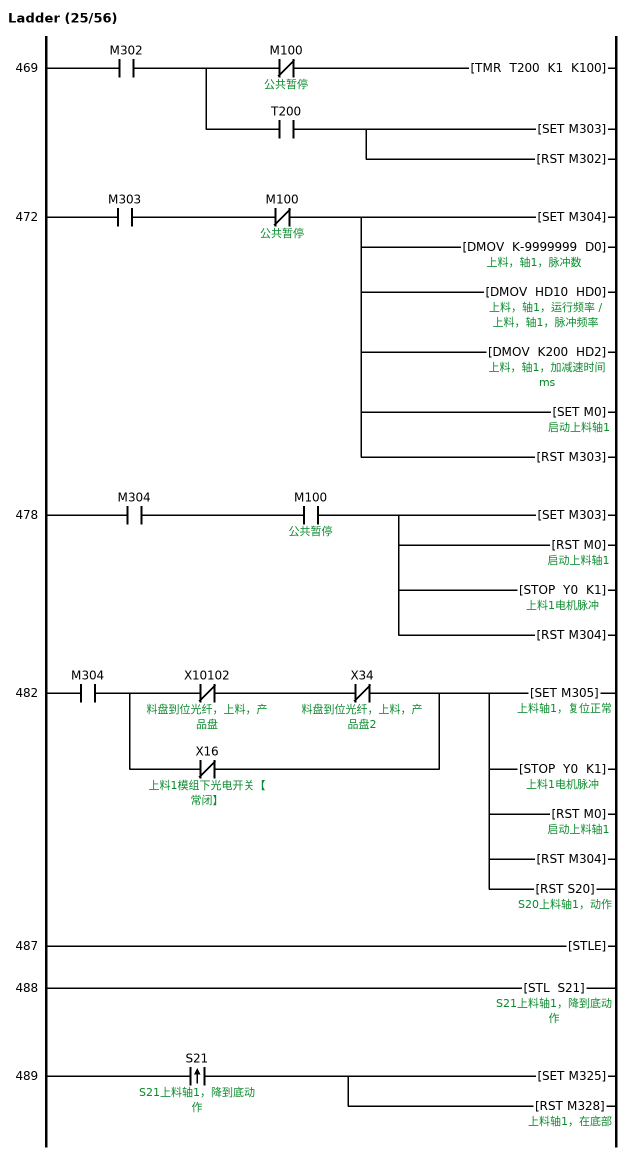
[picture p24: Ladder rows 469-489]
LD     M302
MPS
ANI    M100	; 公共暂停
TMR    T200 K1 K100
MPP
AND    T200
SET    M303
RST    M302
LD     M303
ANI    M100	; 公共暂停
SET    M304
DMOV   K-9999999 D0	; 上料，轴1，脉冲数
DMOV   HD10 HD0	; 上料，轴1，运行频率 / 上料，轴1，脉冲频率
DMOV   K200 HD2	; 上料，轴1，加减速时间ms
SET    M0	; 启动上料轴1
RST    M303
LD     M304
AND    M100	; 公共暂停
SET    M303
RST    M0	; 启动上料轴1
STOP   Y0 K1	; 上料1电机脉冲
RST    M304
LD     M304
LDI    X10102	; 料盘到位光纤，上料，产品盘
ANI    X34	; 料盘到位光纤，上料，产品盘2
ORI    X16	; 上料1模组下光电开关【常闭】
ANB
SET    M305	; 上料轴1，复位正常
STOP   Y0 K1	; 上料1电机脉冲
RST    M0	; 启动上料轴1
RST    M304
RST    S20	; S20上料轴1，动作
STLE
STL    S21	; S21上料轴1，降到底动作
LDP    S21	; S21上料轴1，降到底动作
SET    M325
RST    M328	; 上料轴1，在底部

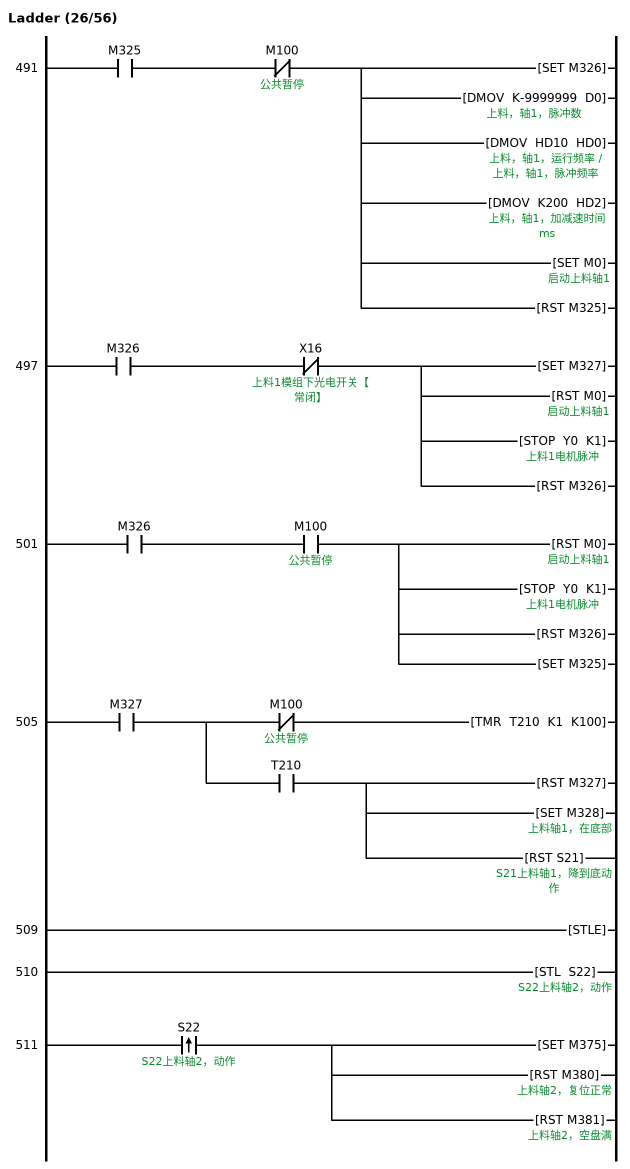
LD     M325
ANI    M100	; 公共暂停
SET    M326
DMOV   K-9999999 D0	; 上料，轴1，脉冲数
DMOV   HD10 HD0	; 上料，轴1，运行频率 / 上料，轴1，脉冲频率
DMOV   K200 HD2	; 上料，轴1，加减速时间ms
SET    M0	; 启动上料轴1
RST    M325
LD     M326
ANI    X16	; 上料1模组下光电开关【常闭】
SET    M327
RST    M0	; 启动上料轴1
STOP   Y0 K1	; 上料1电机脉冲
RST    M326
LD     M326
AND    M100	; 公共暂停
RST    M0	; 启动上料轴1
STOP   Y0 K1	; 上料1电机脉冲
RST    M326
SET    M325
LD     M327
MPS
ANI    M100	; 公共暂停
TMR    T210 K1 K100
MPP
AND    T210
RST    M327
SET    M328	; 上料轴1，在底部
RST    S21	; S21上料轴1，降到底动作
STLE
STL    S22	; S22上料轴2，动作
LDP    S22	; S22上料轴2，动作
SET    M375
RST    M380	; 上料轴2，复位正常
RST    M381	; 上料轴2，空盘满

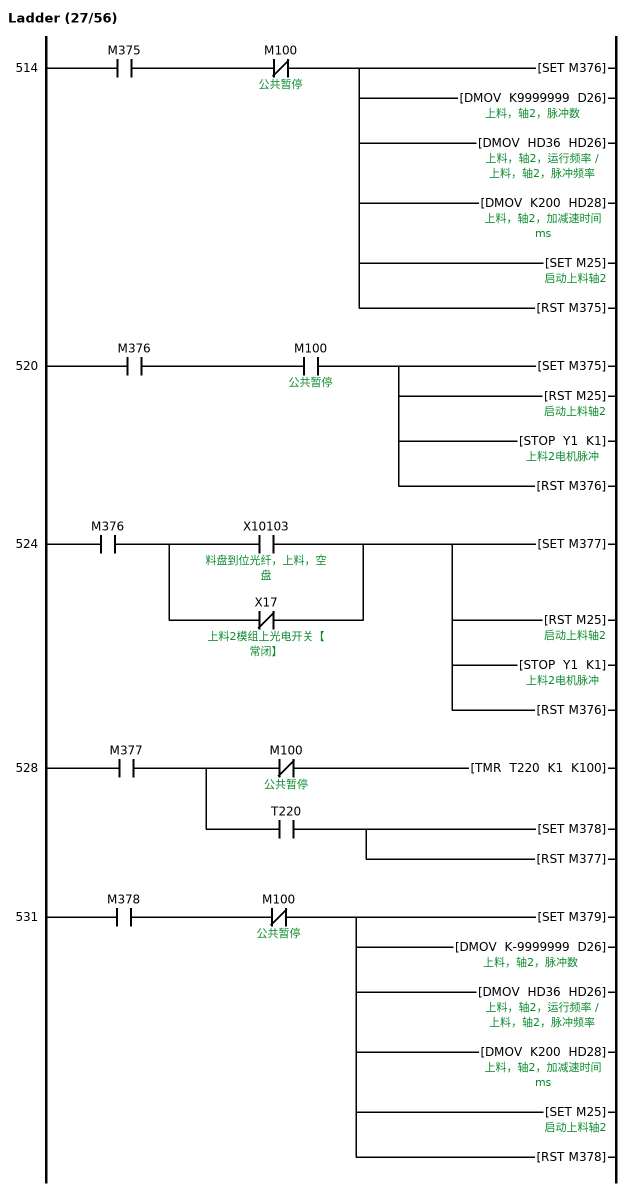
LD     M375
ANI    M100	; 公共暂停
SET    M376
DMOV   K9999999 D26	; 上料，轴2，脉冲数
DMOV   HD36 HD26	; 上料，轴2，运行频率 / 上料，轴2，脉冲频率
DMOV   K200 HD28	; 上料，轴2，加减速时间ms
SET    M25	; 启动上料轴2
RST    M375
LD     M376
AND    M100	; 公共暂停
SET    M375
RST    M25	; 启动上料轴2
STOP   Y1 K1	; 上料2电机脉冲
RST    M376
LD     M376
LD     X10103	; 料盘到位光纤，上料，空盘
ORI    X17	; 上料2模组上光电开关【常闭】
ANB
SET    M377
RST    M25	; 启动上料轴2
STOP   Y1 K1	; 上料2电机脉冲
RST    M376
LD     M377
MPS
ANI    M100	; 公共暂停
TMR    T220 K1 K100
MPP
AND    T220
SET    M378
RST    M377
LD     M378
ANI    M100	; 公共暂停
SET    M379
DMOV   K-9999999 D26	; 上料，轴2，脉冲数
DMOV   HD36 HD26	; 上料，轴2，运行频率 / 上料，轴2，脉冲频率
DMOV   K200 HD28	; 上料，轴2，加减速时间ms
SET    M25	; 启动上料轴2
RST    M378

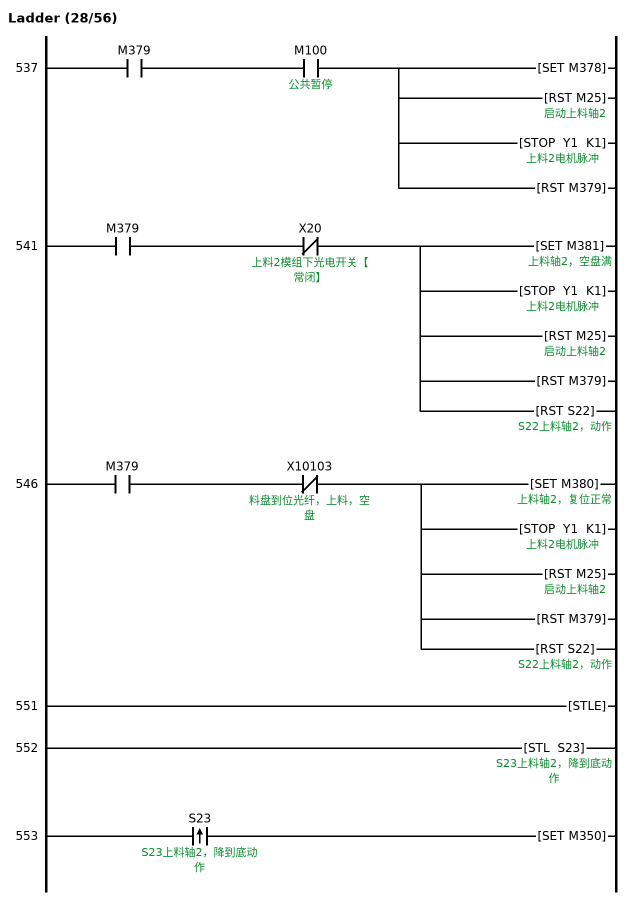
LD     M379
AND    M100	; 公共暂停
SET    M378
RST    M25	; 启动上料轴2
STOP   Y1 K1	; 上料2电机脉冲
RST    M379
LD     M379
ANI    X20	; 上料2模组下光电开关【常闭】
SET    M381	; 上料轴2，空盘满
STOP   Y1 K1	; 上料2电机脉冲
RST    M25	; 启动上料轴2
RST    M379
RST    S22	; S22上料轴2，动作
LD     M379
ANI    X10103	; 料盘到位光纤，上料，空盘
SET    M380	; 上料轴2，复位正常
STOP   Y1 K1	; 上料2电机脉冲
RST    M25	; 启动上料轴2
RST    M379
RST    S22	; S22上料轴2，动作
STLE
STL    S23	; S23上料轴2，降到底动作
LDP    S23	; S23上料轴2，降到底动作
SET    M350

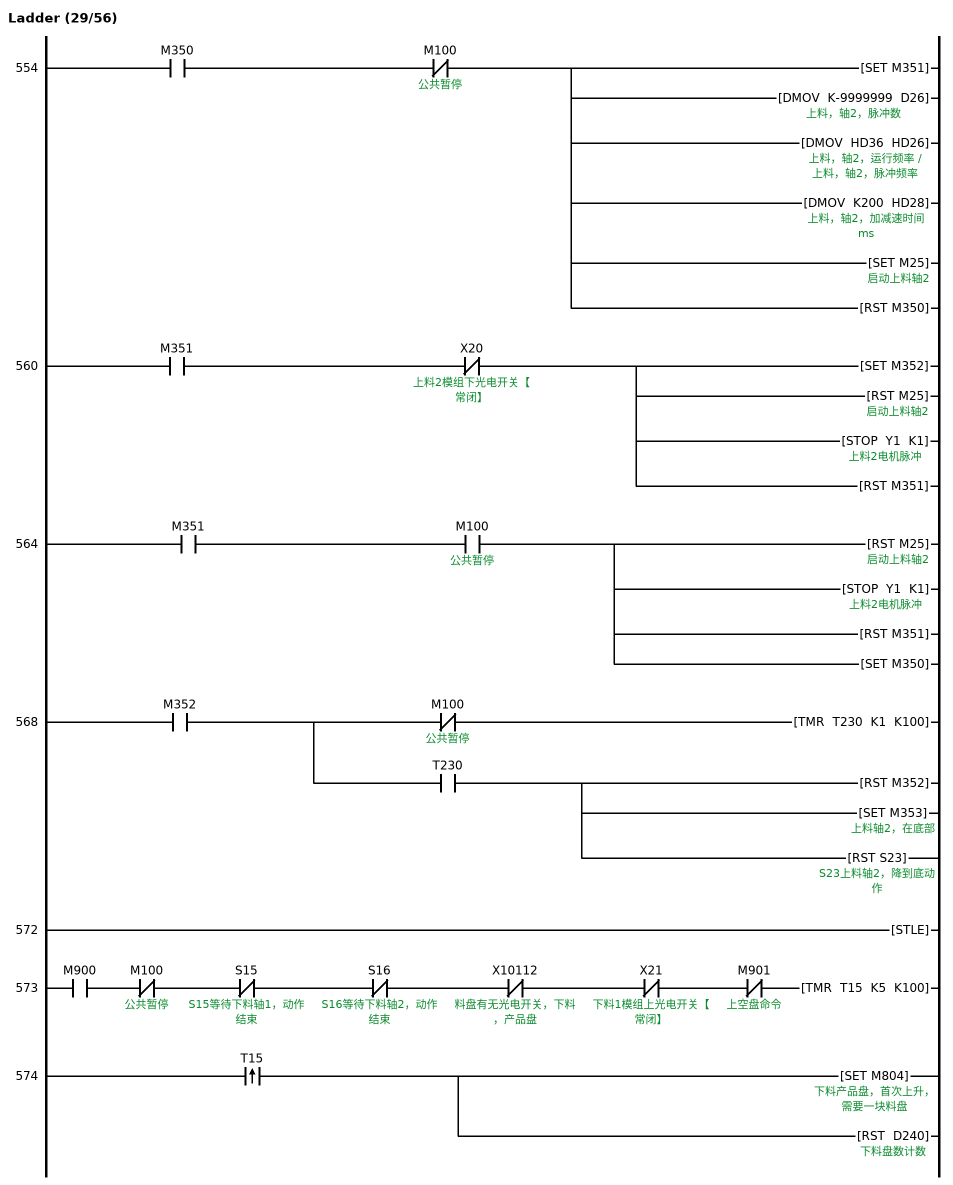
LD     M350
ANI    M100	; 公共暂停
SET    M351
DMOV   K-9999999 D26	; 上料，轴2，脉冲数
DMOV   HD36 HD26	; 上料，轴2，运行频率 / 上料，轴2，脉冲频率
DMOV   K200 HD28	; 上料，轴2，加减速时间ms
SET    M25	; 启动上料轴2
RST    M350
LD     M351
ANI    X20	; 上料2模组下光电开关【常闭】
SET    M352
RST    M25	; 启动上料轴2
STOP   Y1 K1	; 上料2电机脉冲
RST    M351
LD     M351
AND    M100	; 公共暂停
RST    M25	; 启动上料轴2
STOP   Y1 K1	; 上料2电机脉冲
RST    M351
SET    M350
LD     M352
MPS
ANI    M100	; 公共暂停
TMR    T230 K1 K100
MPP
AND    T230
RST    M352
SET    M353	; 上料轴2，在底部
RST    S23	; S23上料轴2，降到底动作
STLE
LD     M900
ANI    M100	; 公共暂停
ANI    S15	; S15等待下料轴1，动作结束
ANI    S16	; S16等待下料轴2，动作结束
ANI    X10112	; 料盘有无光电开关，下料，产品盘
ANI    X21	; 下料1模组上光电开关【常闭】
ANI    M901	; 上空盘命令
TMR    T15 K5 K100
LDP    T15
SET    M804	; 下料产品盘，首次上升，需要一块料盘
RST    D240	; 下料盘数计数

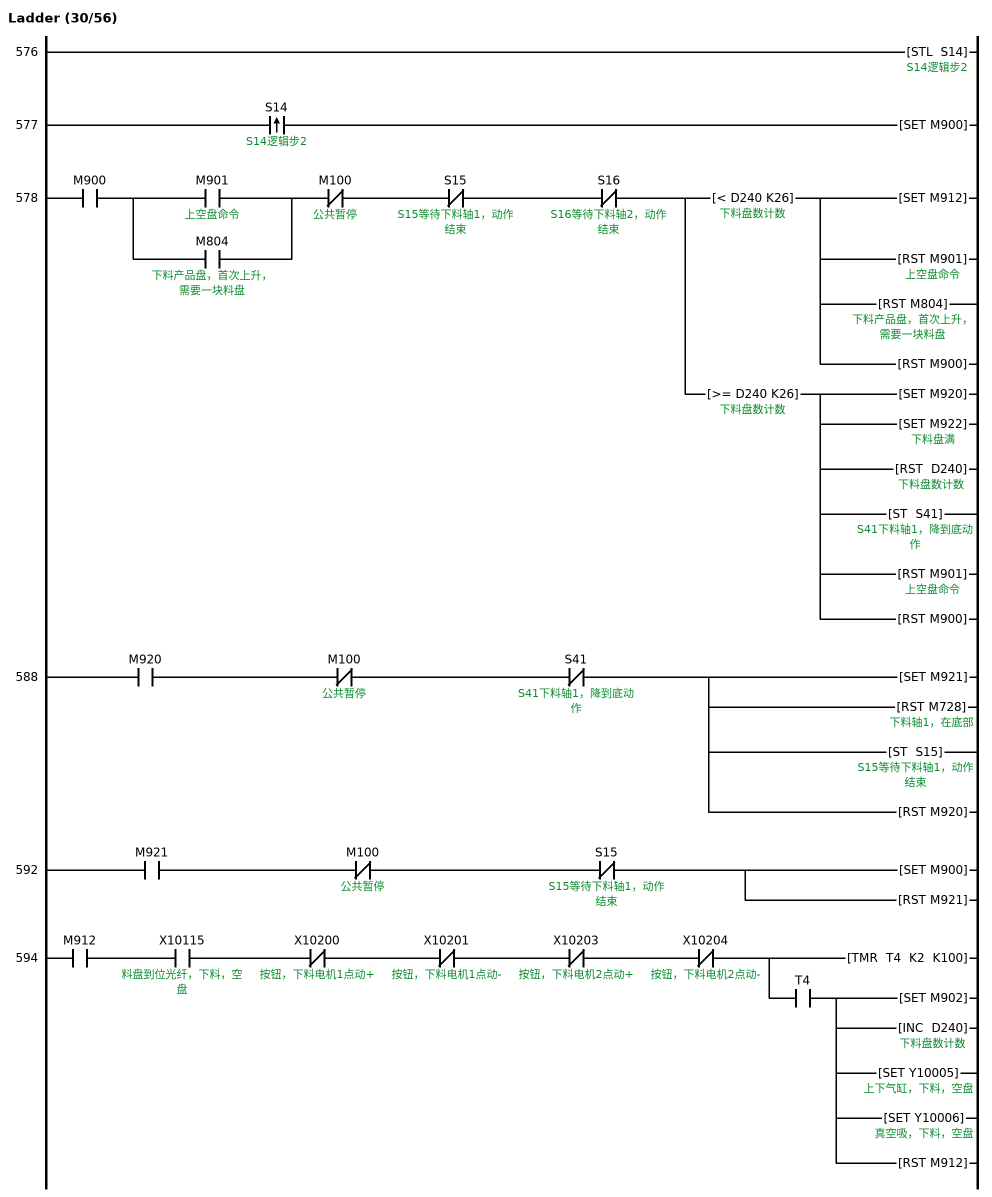
STL    S14	; S14逻辑步2
LDP    S14	; S14逻辑步2
SET    M900
LD     M900
LD     M901	; 上空盘命令
OR     M804	; 下料产品盘，首次上升，需要一块料盘
ANB
ANI    M100	; 公共暂停
ANI    S15	; S15等待下料轴1，动作结束
ANI    S16	; S16等待下料轴2，动作结束
MPS
AND<   D240 K26	; 下料盘数计数
SET    M912
RST    M901	; 上空盘命令
RST    M804	; 下料产品盘，首次上升，需要一块料盘
RST    M900
MPP
AND>=  D240 K26	; 下料盘数计数
SET    M920
SET    M922	; 下料盘满
RST    D240	; 下料盘数计数
ST     S41	; S41下料轴1，降到底动作
RST    M901	; 上空盘命令
RST    M900
LD     M920
ANI    M100	; 公共暂停
ANI    S41	; S41下料轴1，降到底动作
SET    M921
RST    M728	; 下料轴1，在底部
ST     S15	; S15等待下料轴1，动作结束
RST    M920
LD     M921
ANI    M100	; 公共暂停
ANI    S15	; S15等待下料轴1，动作结束
SET    M900
RST    M921
LD     M912
AND    X10115	; 料盘到位光纤，下料，空盘
ANI    X10200	; 按钮，下料电机1点动+
ANI    X10201	; 按钮，下料电机1点动-
ANI    X10203	; 按钮，下料电机2点动+
ANI    X10204	; 按钮，下料电机2点动-
TMR    T4 K2 K100
AND    T4
SET    M902
INC    D240	; 下料盘数计数
SET    Y10005	; 上下气缸，下料，空盘
SET    Y10006	; 真空吸，下料，空盘
RST    M912

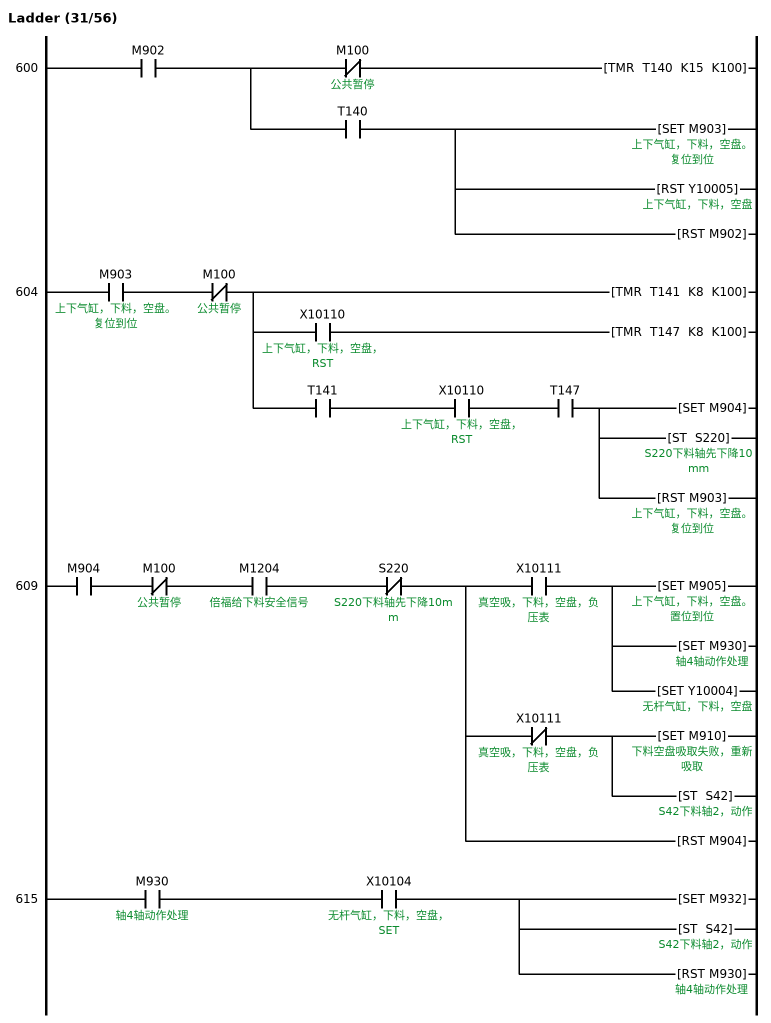
LD     M902
MPS
ANI    M100	; 公共暂停
TMR    T140 K15 K100
MPP
AND    T140
SET    M903	; 上下气缸，下料，空盘。复位到位
RST    Y10005	; 上下气缸，下料，空盘
RST    M902
LD     M903	; 上下气缸，下料，空盘。复位到位
ANI    M100	; 公共暂停
TMR    T141 K8 K100
MPS
AND    X10110	; 上下气缸，下料，空盘，RST
TMR    T147 K8 K100
MPP
AND    T141
AND    X10110	; 上下气缸，下料，空盘，RST
AND    T147
SET    M904
ST     S220	; S220下料轴先下降10mm
RST    M903	; 上下气缸，下料，空盘。复位到位
LD     M904
ANI    M100	; 公共暂停
AND    M1204	; 倍福给下料安全信号
ANI    S220	; S220下料轴先下降10mm
MPS
AND    X10111	; 真空吸，下料，空盘，负压表
SET    M905	; 上下气缸，下料，空盘。置位到位
SET    M930	; 轴4轴动作处理
SET    Y10004	; 无杆气缸，下料，空盘
MRD
ANI    X10111	; 真空吸，下料，空盘，负压表
SET    M910	; 下料空盘吸取失败，重新吸取
ST     S42	; S42下料轴2，动作
MPP
RST    M904
LD     M930	; 轴4轴动作处理
AND    X10104	; 无杆气缸，下料，空盘，SET
SET    M932
ST     S42	; S42下料轴2，动作
RST    M930	; 轴4轴动作处理

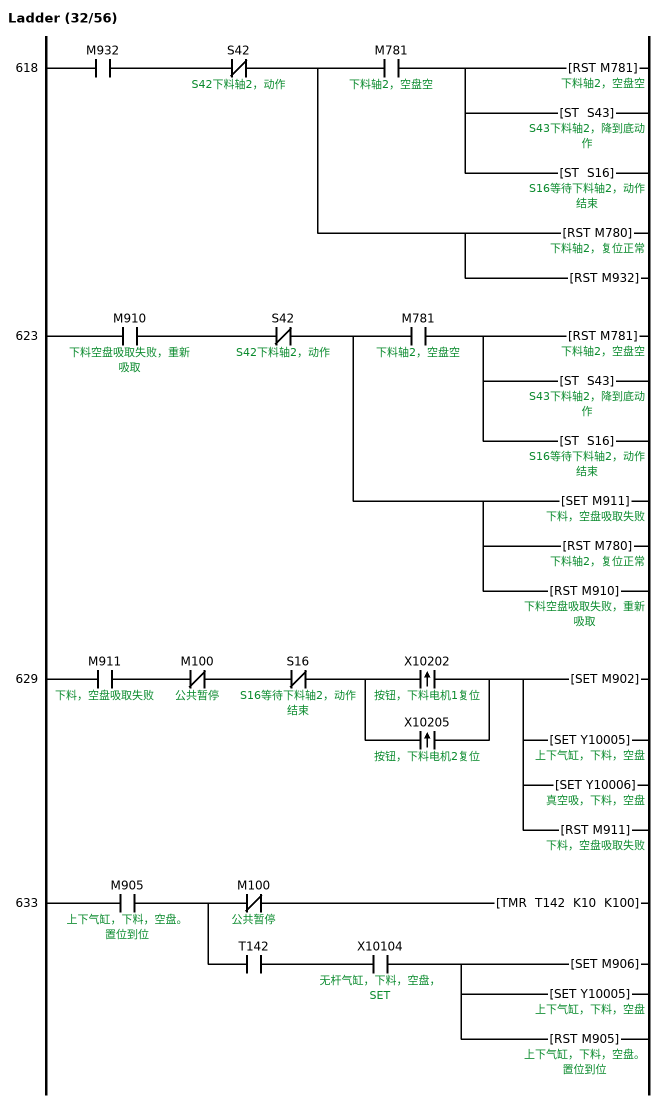
LD     M932
ANI    S42	; S42下料轴2，动作
MPS
AND    M781	; 下料轴2，空盘空
RST    M781	; 下料轴2，空盘空
ST     S43	; S43下料轴2，降到底动作
ST     S16	; S16等待下料轴2，动作结束
MPP
RST    M780	; 下料轴2，复位正常
RST    M932
LD     M910	; 下料空盘吸取失败，重新吸取
ANI    S42	; S42下料轴2，动作
MPS
AND    M781	; 下料轴2，空盘空
RST    M781	; 下料轴2，空盘空
ST     S43	; S43下料轴2，降到底动作
ST     S16	; S16等待下料轴2，动作结束
MPP
SET    M911	; 下料，空盘吸取失败
RST    M780	; 下料轴2，复位正常
RST    M910	; 下料空盘吸取失败，重新吸取
LD     M911	; 下料，空盘吸取失败
ANI    M100	; 公共暂停
ANI    S16	; S16等待下料轴2，动作结束
LDP    X10202	; 按钮，下料电机1复位
ORP    X10205	; 按钮，下料电机2复位
ANB
SET    M902
SET    Y10005	; 上下气缸，下料，空盘
SET    Y10006	; 真空吸，下料，空盘
RST    M911	; 下料，空盘吸取失败
LD     M905	; 上下气缸，下料，空盘。置位到位
MPS
ANI    M100	; 公共暂停
TMR    T142 K10 K100
MPP
AND    T142
AND    X10104	; 无杆气缸，下料，空盘，SET
SET    M906
SET    Y10005	; 上下气缸，下料，空盘
RST    M905	; 上下气缸，下料，空盘。置位到位

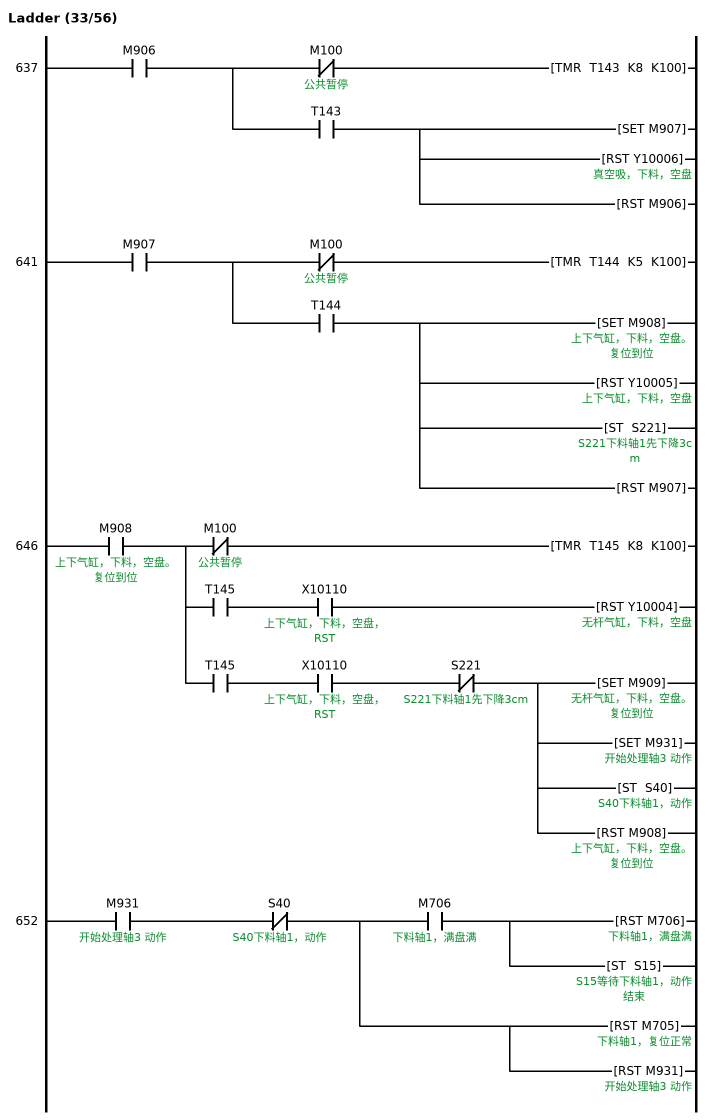
LD     M906
MPS
ANI    M100	; 公共暂停
TMR    T143 K8 K100
MPP
AND    T143
SET    M907
RST    Y10006	; 真空吸，下料，空盘
RST    M906
LD     M907
MPS
ANI    M100	; 公共暂停
TMR    T144 K5 K100
MPP
AND    T144
SET    M908	; 上下气缸，下料，空盘。复位到位
RST    Y10005	; 上下气缸，下料，空盘
ST     S221	; S221下料轴1先下降3cm
RST    M907
LD     M908	; 上下气缸，下料，空盘。复位到位
MPS
ANI    M100	; 公共暂停
TMR    T145 K8 K100
MRD
AND    T145
AND    X10110	; 上下气缸，下料，空盘，RST
RST    Y10004	; 无杆气缸，下料，空盘
MPP
AND    T145
AND    X10110	; 上下气缸，下料，空盘，RST
ANI    S221	; S221下料轴1先下降3cm
SET    M909	; 无杆气缸，下料，空盘。复位到位
SET    M931	; 开始处理轴3 动作
ST     S40	; S40下料轴1，动作
RST    M908	; 上下气缸，下料，空盘。复位到位
LD     M931	; 开始处理轴3 动作
ANI    S40	; S40下料轴1，动作
MPS
AND    M706	; 下料轴1，满盘满
RST    M706	; 下料轴1，满盘满
ST     S15	; S15等待下料轴1，动作结束
MPP
RST    M705	; 下料轴1，复位正常
RST    M931	; 开始处理轴3 动作

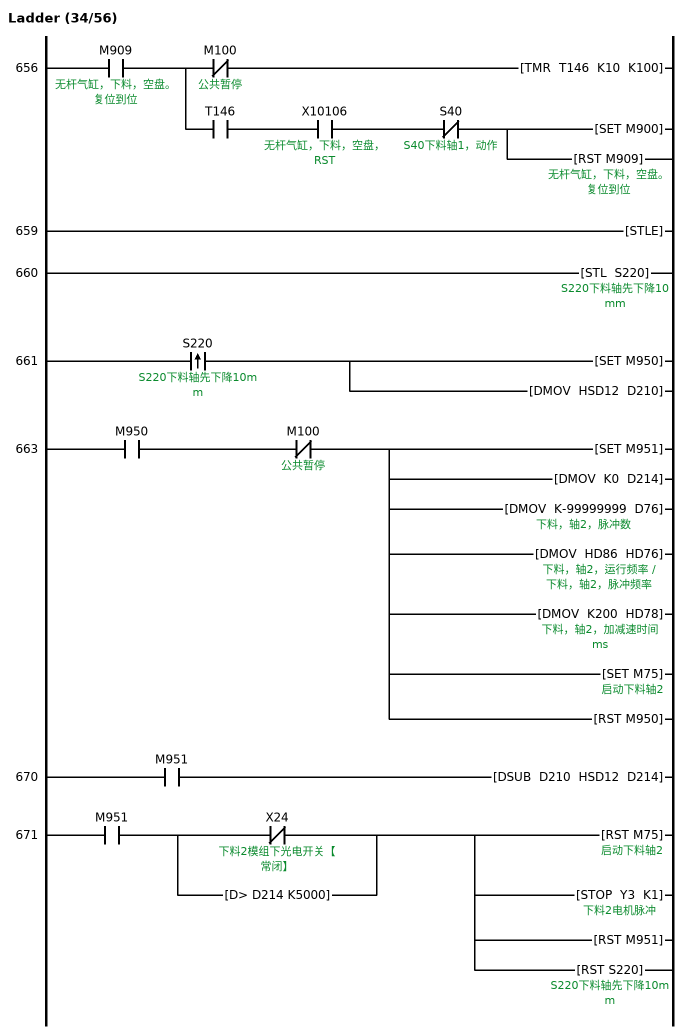
LD     M909	; 无杆气缸，下料，空盘。复位到位
MPS
ANI    M100	; 公共暂停
TMR    T146 K10 K100
MPP
AND    T146
AND    X10106	; 无杆气缸，下料，空盘，RST
ANI    S40	; S40下料轴1，动作
SET    M900
RST    M909	; 无杆气缸，下料，空盘。复位到位
STLE
STL    S220	; S220下料轴先下降10mm
LDP    S220	; S220下料轴先下降10mm
SET    M950
DMOV   HSD12 D210
LD     M950
ANI    M100	; 公共暂停
SET    M951
DMOV   K0 D214
DMOV   K-99999999 D76	; 下料，轴2，脉冲数
DMOV   HD86 HD76	; 下料，轴2，运行频率 / 下料，轴2，脉冲频率
DMOV   K200 HD78	; 下料，轴2，加减速时间ms
SET    M75	; 启动下料轴2
RST    M950
LD     M951
DSUB   D210 HSD12 D214
LD     M951
LDI    X24	; 下料2模组下光电开关【常闭】
DOR>   D214 K5000
ANB
RST    M75	; 启动下料轴2
STOP   Y3 K1	; 下料2电机脉冲
RST    M951
RST    S220	; S220下料轴先下降10mm

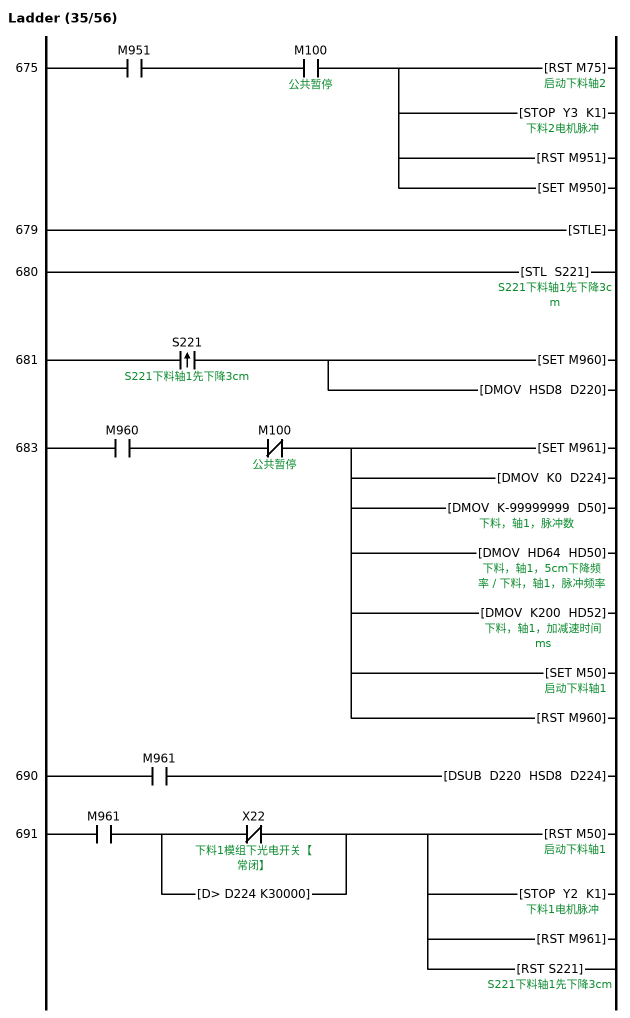
LD     M951
AND    M100	; 公共暂停
RST    M75	; 启动下料轴2
STOP   Y3 K1	; 下料2电机脉冲
RST    M951
SET    M950
STLE
STL    S221	; S221下料轴1先下降3cm
LDP    S221	; S221下料轴1先下降3cm
SET    M960
DMOV   HSD8 D220
LD     M960
ANI    M100	; 公共暂停
SET    M961
DMOV   K0 D224
DMOV   K-99999999 D50	; 下料，轴1，脉冲数
DMOV   HD64 HD50	; 下料，轴1，5cm下降频率 / 下料，轴1，脉冲频率
DMOV   K200 HD52	; 下料，轴1，加减速时间ms
SET    M50	; 启动下料轴1
RST    M960
LD     M961
DSUB   D220 HSD8 D224
LD     M961
LDI    X22	; 下料1模组下光电开关【常闭】
DOR>   D224 K30000
ANB
RST    M50	; 启动下料轴1
STOP   Y2 K1	; 下料1电机脉冲
RST    M961
RST    S221	; S221下料轴1先下降3cm

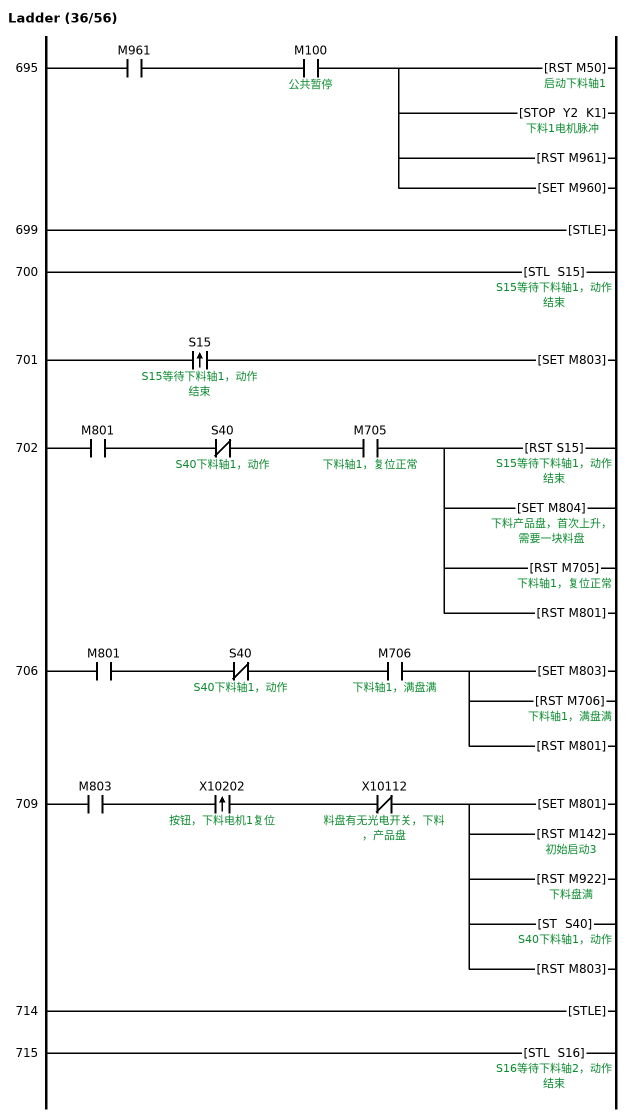
LD     M961
AND    M100	; 公共暂停
RST    M50	; 启动下料轴1
STOP   Y2 K1	; 下料1电机脉冲
RST    M961
SET    M960
STLE
STL    S15	; S15等待下料轴1，动作结束
LDP    S15	; S15等待下料轴1，动作结束
SET    M803
LD     M801
ANI    S40	; S40下料轴1，动作
AND    M705	; 下料轴1，复位正常
RST    S15	; S15等待下料轴1，动作结束
SET    M804	; 下料产品盘，首次上升，需要一块料盘
RST    M705	; 下料轴1，复位正常
RST    M801
LD     M801
ANI    S40	; S40下料轴1，动作
AND    M706	; 下料轴1，满盘满
SET    M803
RST    M706	; 下料轴1，满盘满
RST    M801
LD     M803
ANDP   X10202	; 按钮，下料电机1复位
ANI    X10112	; 料盘有无光电开关，下料，产品盘
SET    M801
RST    M142	; 初始启动3
RST    M922	; 下料盘满
ST     S40	; S40下料轴1，动作
RST    M803
STLE
STL    S16	; S16等待下料轴2，动作结束

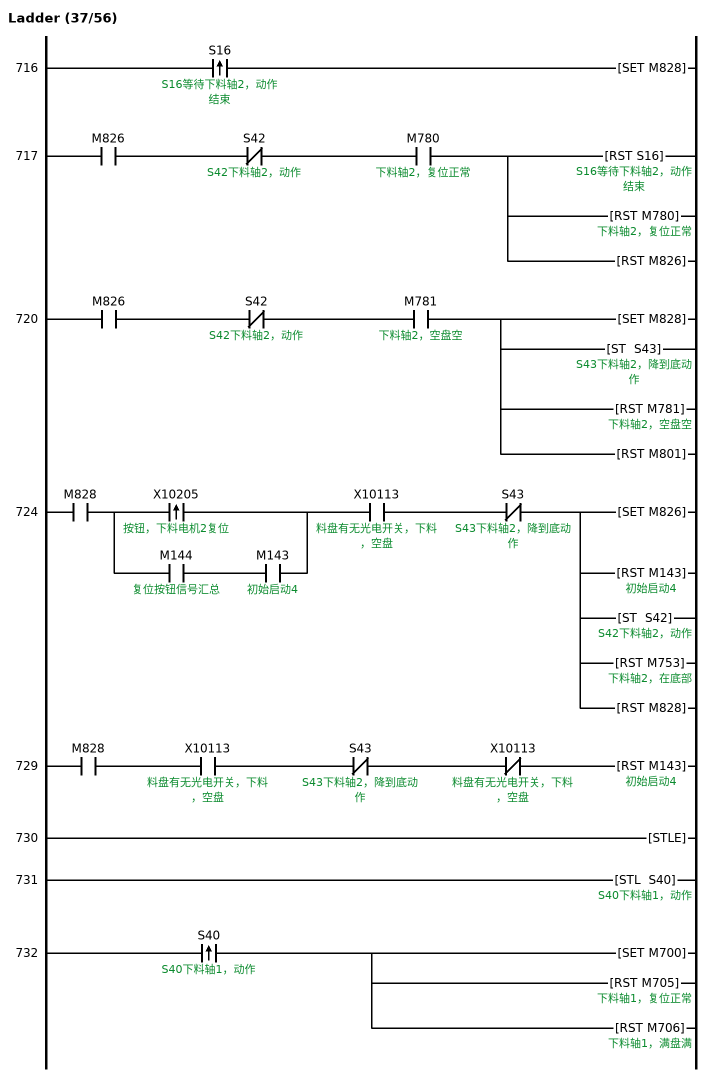
LDP    S16	; S16等待下料轴2，动作结束
SET    M828
LD     M826
ANI    S42	; S42下料轴2，动作
AND    M780	; 下料轴2，复位正常
RST    S16	; S16等待下料轴2，动作结束
RST    M780	; 下料轴2，复位正常
RST    M826
LD     M826
ANI    S42	; S42下料轴2，动作
AND    M781	; 下料轴2，空盘空
SET    M828
ST     S43	; S43下料轴2，降到底动作
RST    M781	; 下料轴2，空盘空
RST    M801
LD     M828
LDP    X10205	; 按钮，下料电机2复位
LD     M144	; 复位按钮信号汇总
AND    M143	; 初始启动4
ORB
ANB
AND    X10113	; 料盘有无光电开关，下料，空盘
ANI    S43	; S43下料轴2，降到底动作
SET    M826
RST    M143	; 初始启动4
ST     S42	; S42下料轴2，动作
RST    M753	; 下料轴2，在底部
RST    M828
LD     M828
AND    X10113	; 料盘有无光电开关，下料，空盘
ANI    S43	; S43下料轴2，降到底动作
ANI    X10113	; 料盘有无光电开关，下料，空盘
RST    M143	; 初始启动4
STLE
STL    S40	; S40下料轴1，动作
LDP    S40	; S40下料轴1，动作
SET    M700
RST    M705	; 下料轴1，复位正常
RST    M706	; 下料轴1，满盘满

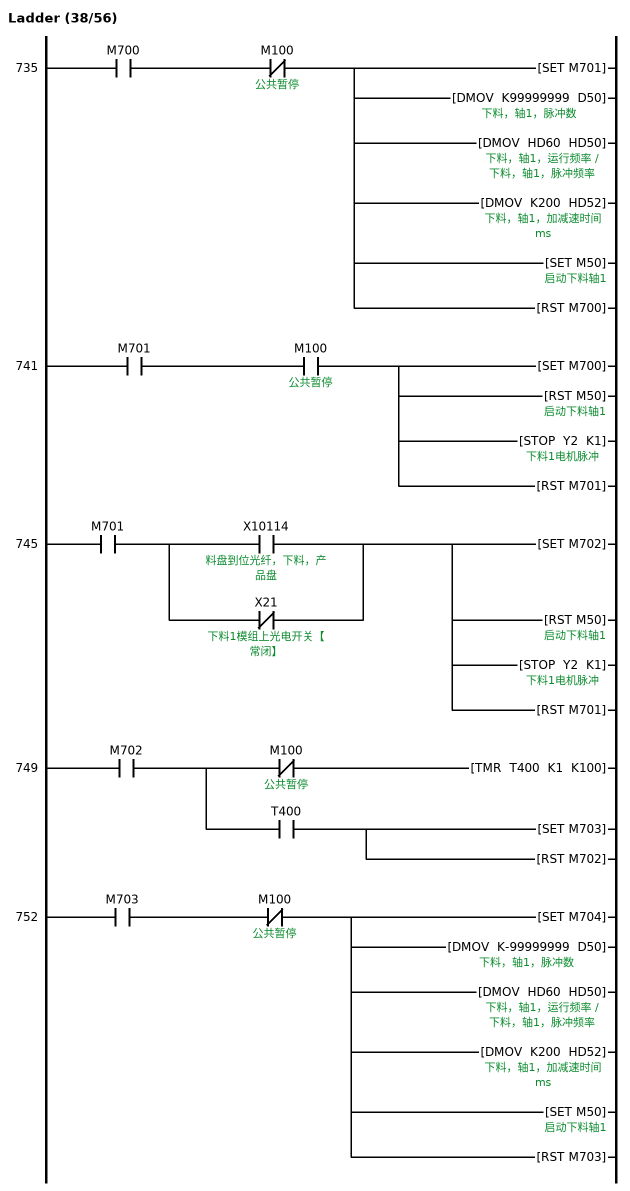
LD     M700
ANI    M100	; 公共暂停
SET    M701
DMOV   K99999999 D50	; 下料，轴1，脉冲数
DMOV   HD60 HD50	; 下料，轴1，运行频率 / 下料，轴1，脉冲频率
DMOV   K200 HD52	; 下料，轴1，加减速时间ms
SET    M50	; 启动下料轴1
RST    M700
LD     M701
AND    M100	; 公共暂停
SET    M700
RST    M50	; 启动下料轴1
STOP   Y2 K1	; 下料1电机脉冲
RST    M701
LD     M701
LD     X10114	; 料盘到位光纤，下料，产品盘
ORI    X21	; 下料1模组上光电开关【常闭】
ANB
SET    M702
RST    M50	; 启动下料轴1
STOP   Y2 K1	; 下料1电机脉冲
RST    M701
LD     M702
MPS
ANI    M100	; 公共暂停
TMR    T400 K1 K100
MPP
AND    T400
SET    M703
RST    M702
LD     M703
ANI    M100	; 公共暂停
SET    M704
DMOV   K-99999999 D50	; 下料，轴1，脉冲数
DMOV   HD60 HD50	; 下料，轴1，运行频率 / 下料，轴1，脉冲频率
DMOV   K200 HD52	; 下料，轴1，加减速时间ms
SET    M50	; 启动下料轴1
RST    M703

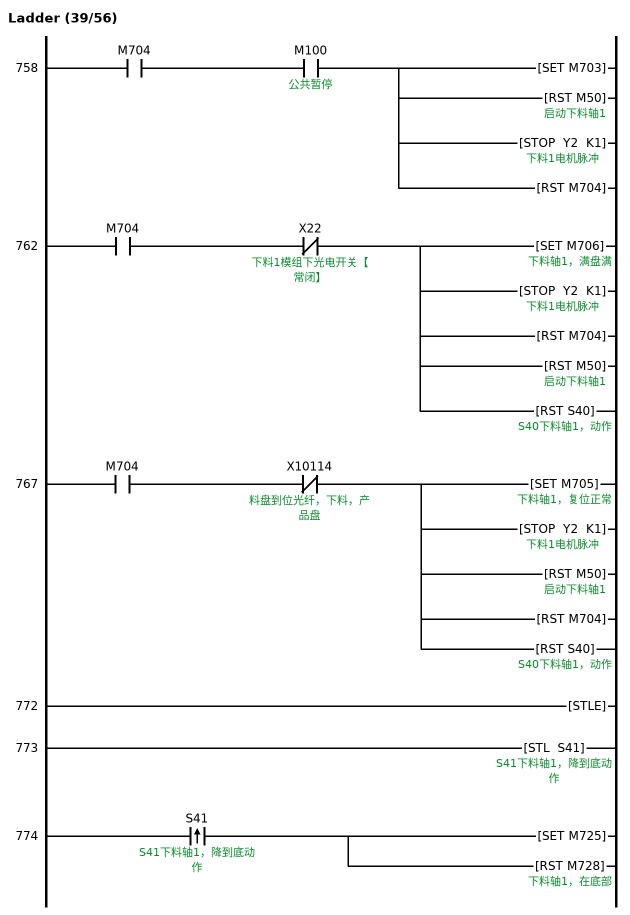
LD     M704
AND    M100	; 公共暂停
SET    M703
RST    M50	; 启动下料轴1
STOP   Y2 K1	; 下料1电机脉冲
RST    M704
LD     M704
ANI    X22	; 下料1模组下光电开关【常闭】
SET    M706	; 下料轴1，满盘满
STOP   Y2 K1	; 下料1电机脉冲
RST    M704
RST    M50	; 启动下料轴1
RST    S40	; S40下料轴1，动作
LD     M704
ANI    X10114	; 料盘到位光纤，下料，产品盘
SET    M705	; 下料轴1，复位正常
STOP   Y2 K1	; 下料1电机脉冲
RST    M50	; 启动下料轴1
RST    M704
RST    S40	; S40下料轴1，动作
STLE
STL    S41	; S41下料轴1，降到底动作
LDP    S41	; S41下料轴1，降到底动作
SET    M725
RST    M728	; 下料轴1，在底部

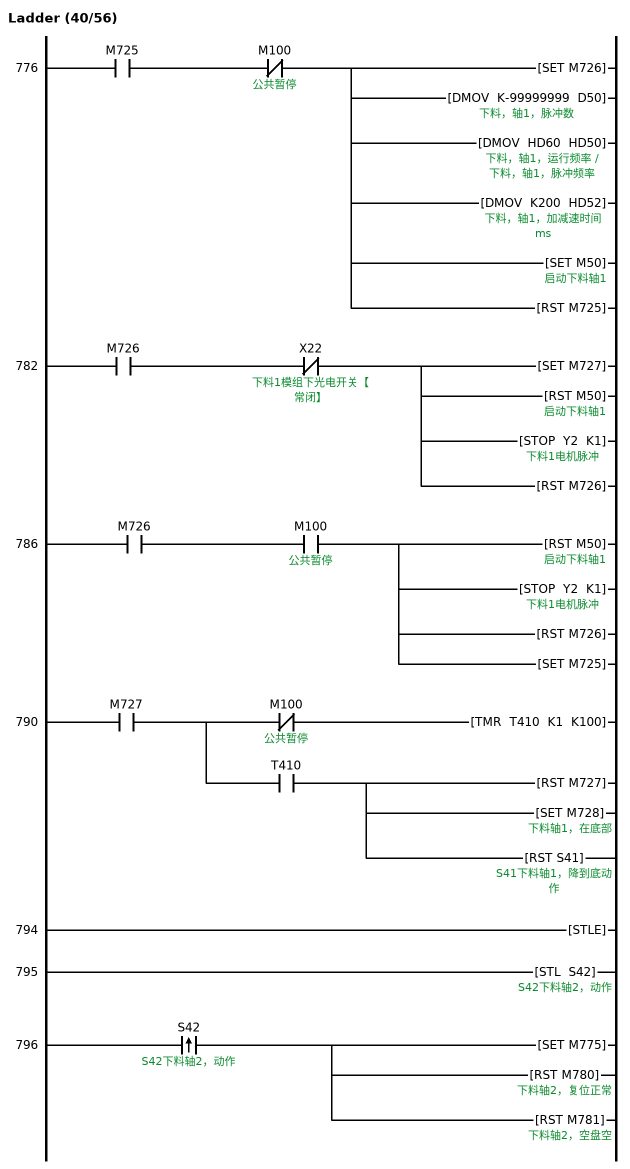
LD     M725
ANI    M100	; 公共暂停
SET    M726
DMOV   K-99999999 D50	; 下料，轴1，脉冲数
DMOV   HD60 HD50	; 下料，轴1，运行频率 / 下料，轴1，脉冲频率
DMOV   K200 HD52	; 下料，轴1，加减速时间ms
SET    M50	; 启动下料轴1
RST    M725
LD     M726
ANI    X22	; 下料1模组下光电开关【常闭】
SET    M727
RST    M50	; 启动下料轴1
STOP   Y2 K1	; 下料1电机脉冲
RST    M726
LD     M726
AND    M100	; 公共暂停
RST    M50	; 启动下料轴1
STOP   Y2 K1	; 下料1电机脉冲
RST    M726
SET    M725
LD     M727
MPS
ANI    M100	; 公共暂停
TMR    T410 K1 K100
MPP
AND    T410
RST    M727
SET    M728	; 下料轴1，在底部
RST    S41	; S41下料轴1，降到底动作
STLE
STL    S42	; S42下料轴2，动作
LDP    S42	; S42下料轴2，动作
SET    M775
RST    M780	; 下料轴2，复位正常
RST    M781	; 下料轴2，空盘空

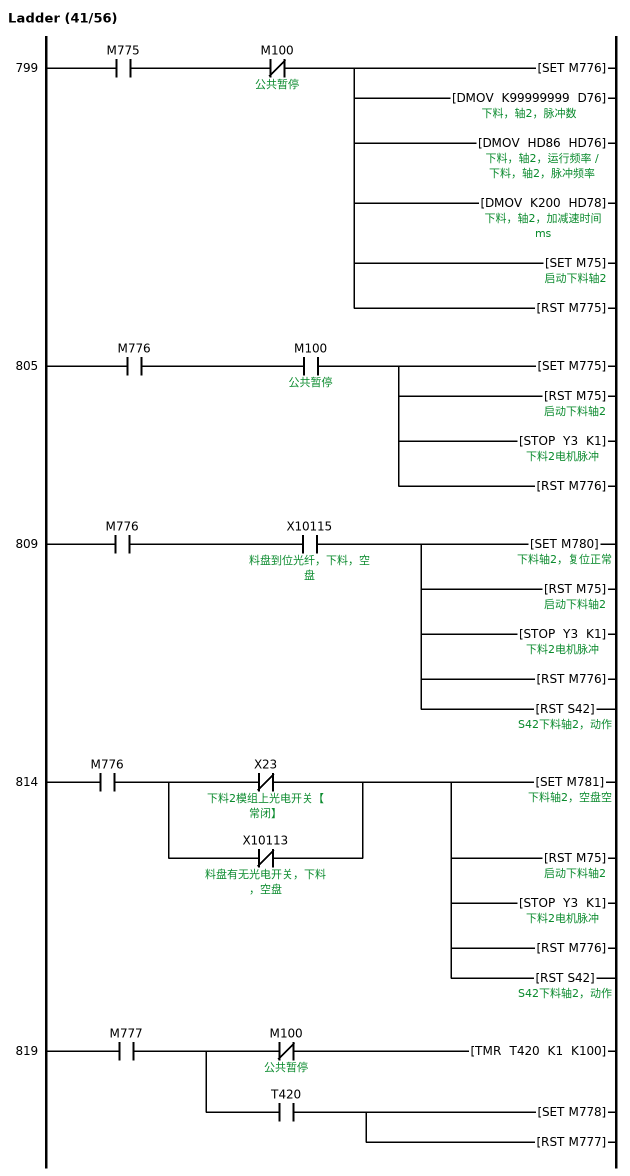
LD     M775
ANI    M100	; 公共暂停
SET    M776
DMOV   K99999999 D76	; 下料，轴2，脉冲数
DMOV   HD86 HD76	; 下料，轴2，运行频率 / 下料，轴2，脉冲频率
DMOV   K200 HD78	; 下料，轴2，加减速时间ms
SET    M75	; 启动下料轴2
RST    M775
LD     M776
AND    M100	; 公共暂停
SET    M775
RST    M75	; 启动下料轴2
STOP   Y3 K1	; 下料2电机脉冲
RST    M776
LD     M776
AND    X10115	; 料盘到位光纤，下料，空盘
SET    M780	; 下料轴2，复位正常
RST    M75	; 启动下料轴2
STOP   Y3 K1	; 下料2电机脉冲
RST    M776
RST    S42	; S42下料轴2，动作
LD     M776
LDI    X23	; 下料2模组上光电开关【常闭】
ORI    X10113	; 料盘有无光电开关，下料，空盘
ANB
SET    M781	; 下料轴2，空盘空
RST    M75	; 启动下料轴2
STOP   Y3 K1	; 下料2电机脉冲
RST    M776
RST    S42	; S42下料轴2，动作
LD     M777
MPS
ANI    M100	; 公共暂停
TMR    T420 K1 K100
MPP
AND    T420
SET    M778
RST    M777

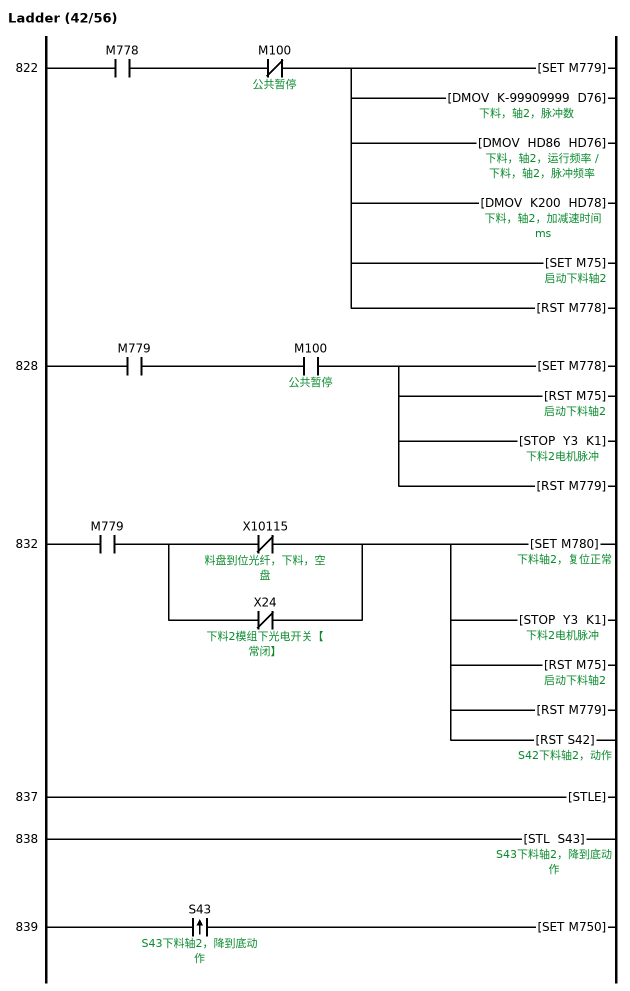
LD     M778
ANI    M100	; 公共暂停
SET    M779
DMOV   K-99909999 D76	; 下料，轴2，脉冲数
DMOV   HD86 HD76	; 下料，轴2，运行频率 / 下料，轴2，脉冲频率
DMOV   K200 HD78	; 下料，轴2，加减速时间ms
SET    M75	; 启动下料轴2
RST    M778
LD     M779
AND    M100	; 公共暂停
SET    M778
RST    M75	; 启动下料轴2
STOP   Y3 K1	; 下料2电机脉冲
RST    M779
LD     M779
LDI    X10115	; 料盘到位光纤，下料，空盘
ORI    X24	; 下料2模组下光电开关【常闭】
ANB
SET    M780	; 下料轴2，复位正常
STOP   Y3 K1	; 下料2电机脉冲
RST    M75	; 启动下料轴2
RST    M779
RST    S42	; S42下料轴2，动作
STLE
STL    S43	; S43下料轴2，降到底动作
LDP    S43	; S43下料轴2，降到底动作
SET    M750

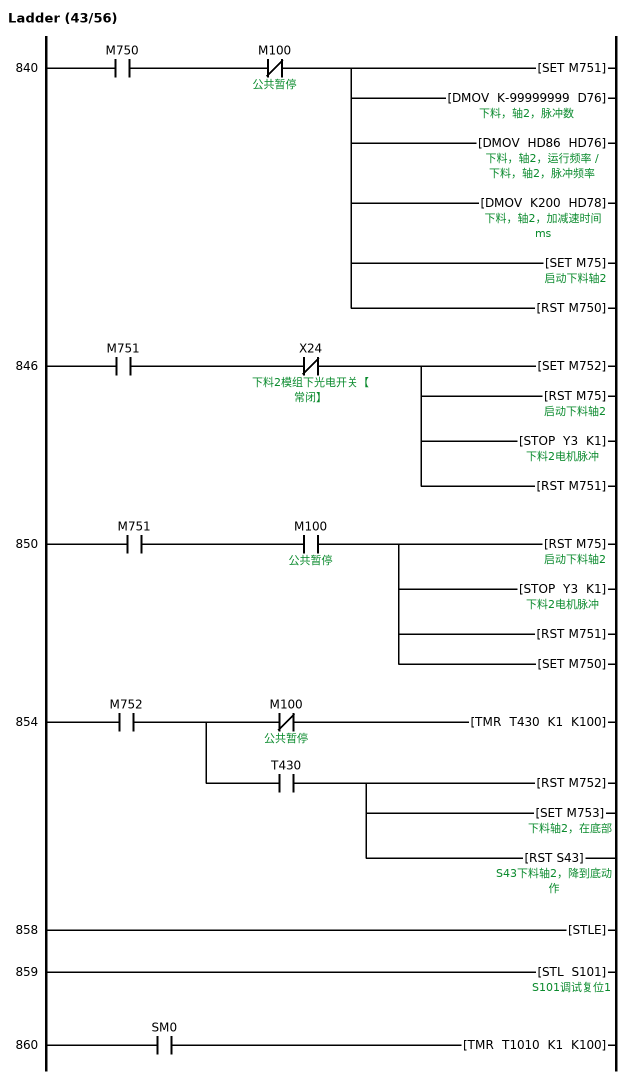
LD     M750
ANI    M100	; 公共暂停
SET    M751
DMOV   K-99999999 D76	; 下料，轴2，脉冲数
DMOV   HD86 HD76	; 下料，轴2，运行频率 / 下料，轴2，脉冲频率
DMOV   K200 HD78	; 下料，轴2，加减速时间ms
SET    M75	; 启动下料轴2
RST    M750
LD     M751
ANI    X24	; 下料2模组下光电开关【常闭】
SET    M752
RST    M75	; 启动下料轴2
STOP   Y3 K1	; 下料2电机脉冲
RST    M751
LD     M751
AND    M100	; 公共暂停
RST    M75	; 启动下料轴2
STOP   Y3 K1	; 下料2电机脉冲
RST    M751
SET    M750
LD     M752
MPS
ANI    M100	; 公共暂停
TMR    T430 K1 K100
MPP
AND    T430
RST    M752
SET    M753	; 下料轴2，在底部
RST    S43	; S43下料轴2，降到底动作
STLE
STL    S101	; S101调试复位1
LD     SM0
TMR    T1010 K1 K100

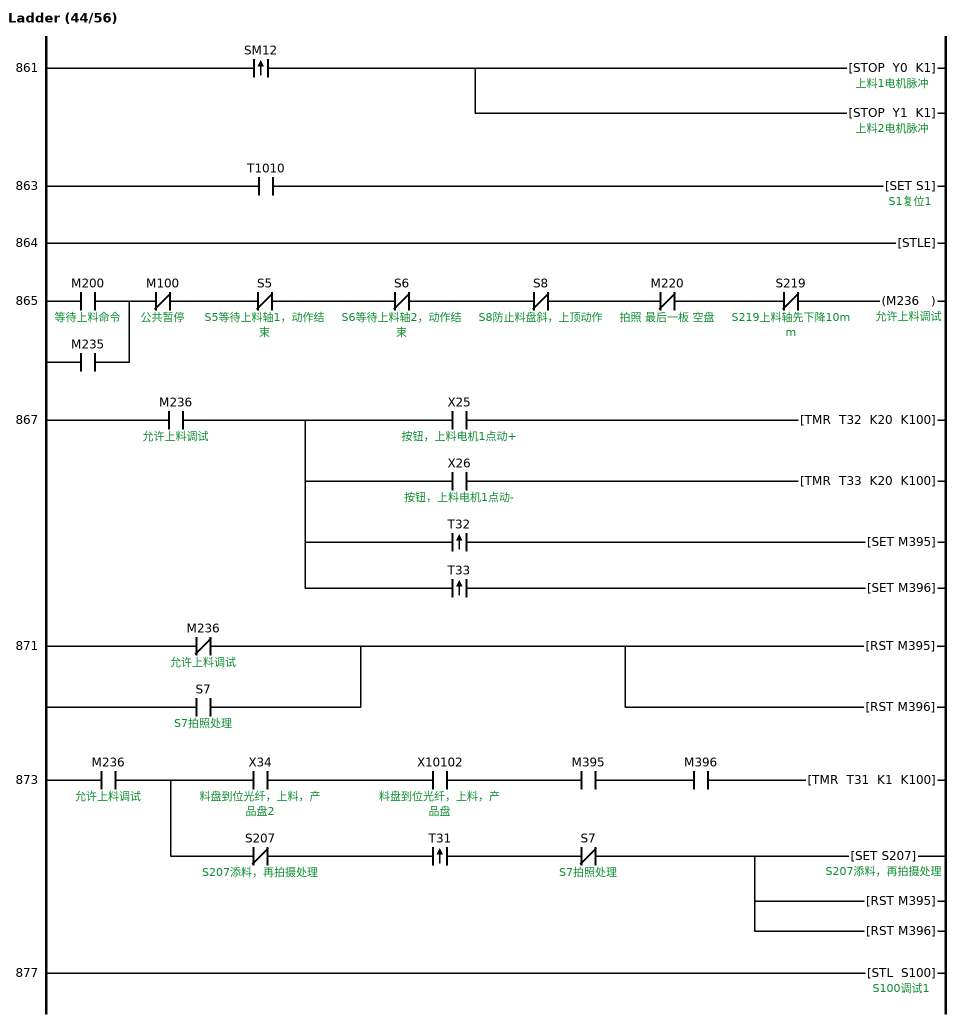
LDP    SM12
STOP   Y0 K1	; 上料1电机脉冲
STOP   Y1 K1	; 上料2电机脉冲
LD     T1010
SET    S1	; S1复位1
STLE
LD     M200	; 等待上料命令
OR     M235
ANI    M100	; 公共暂停
ANI    S5	; S5等待上料轴1，动作结束
ANI    S6	; S6等待上料轴2，动作结束
ANI    S8	; S8防止料盘斜，上顶动作
ANI    M220	; 拍照 最后一板 空盘
ANI    S219	; S219上料轴先下降10mm
OUT    M236	; 允许上料调试
LD     M236	; 允许上料调试
MPS
AND    X25	; 按钮，上料电机1点动+
TMR    T32 K20 K100
MRD
AND    X26	; 按钮，上料电机1点动-
TMR    T33 K20 K100
MRD
ANDP   T32
SET    M395
MPP
ANDP   T33
SET    M396
LDI    M236	; 允许上料调试
OR     S7	; S7拍照处理
RST    M395
RST    M396
LD     M236	; 允许上料调试
MPS
AND    X34	; 料盘到位光纤，上料，产品盘2
AND    X10102	; 料盘到位光纤，上料，产品盘
AND    M395
AND    M396
TMR    T31 K1 K100
MPP
ANI    S207	; S207添料，再拍摄处理
ANDP   T31
ANI    S7	; S7拍照处理
SET    S207	; S207添料，再拍摄处理
RST    M395
RST    M396
STL    S100	; S100调试1

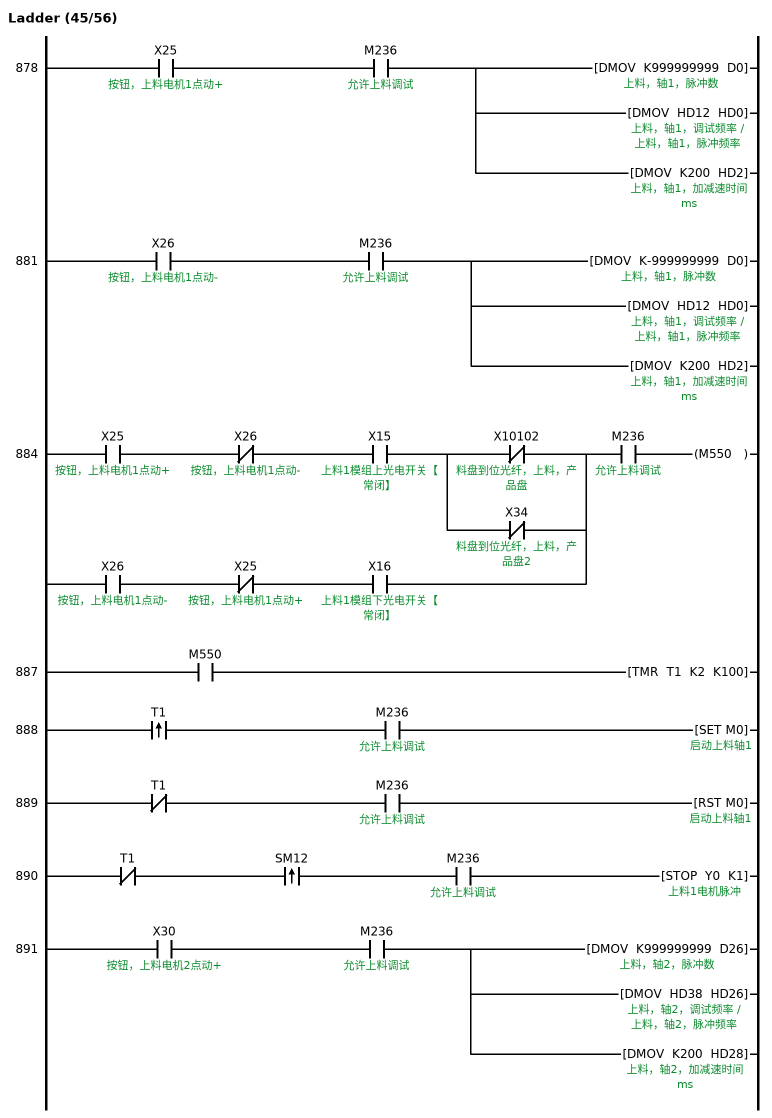
LD     X25	; 按钮，上料电机1点动+
AND    M236	; 允许上料调试
DMOV   K999999999 D0	; 上料，轴1，脉冲数
DMOV   HD12 HD0	; 上料，轴1，调试频率 / 上料，轴1，脉冲频率
DMOV   K200 HD2	; 上料，轴1，加减速时间ms
LD     X26	; 按钮，上料电机1点动-
AND    M236	; 允许上料调试
DMOV   K-999999999 D0	; 上料，轴1，脉冲数
DMOV   HD12 HD0	; 上料，轴1，调试频率 / 上料，轴1，脉冲频率
DMOV   K200 HD2	; 上料，轴1，加减速时间ms
LD     X25	; 按钮，上料电机1点动+
ANI    X26	; 按钮，上料电机1点动-
AND    X15	; 上料1模组上光电开关【常闭】
LDI    X10102	; 料盘到位光纤，上料，产品盘
ORI    X34	; 料盘到位光纤，上料，产品盘2
ANB
LD     X26	; 按钮，上料电机1点动-
ANI    X25	; 按钮，上料电机1点动+
AND    X16	; 上料1模组下光电开关【常闭】
ORB
AND    M236	; 允许上料调试
OUT    M550
LD     M550
TMR    T1 K2 K100
LDP    T1
AND    M236	; 允许上料调试
SET    M0	; 启动上料轴1
LDI    T1
AND    M236	; 允许上料调试
RST    M0	; 启动上料轴1
LDI    T1
ANDP   SM12
AND    M236	; 允许上料调试
STOP   Y0 K1	; 上料1电机脉冲
LD     X30	; 按钮，上料电机2点动+
AND    M236	; 允许上料调试
DMOV   K999999999 D26	; 上料，轴2，脉冲数
DMOV   HD38 HD26	; 上料，轴2，调试频率 / 上料，轴2，脉冲频率
DMOV   K200 HD28	; 上料，轴2，加减速时间ms

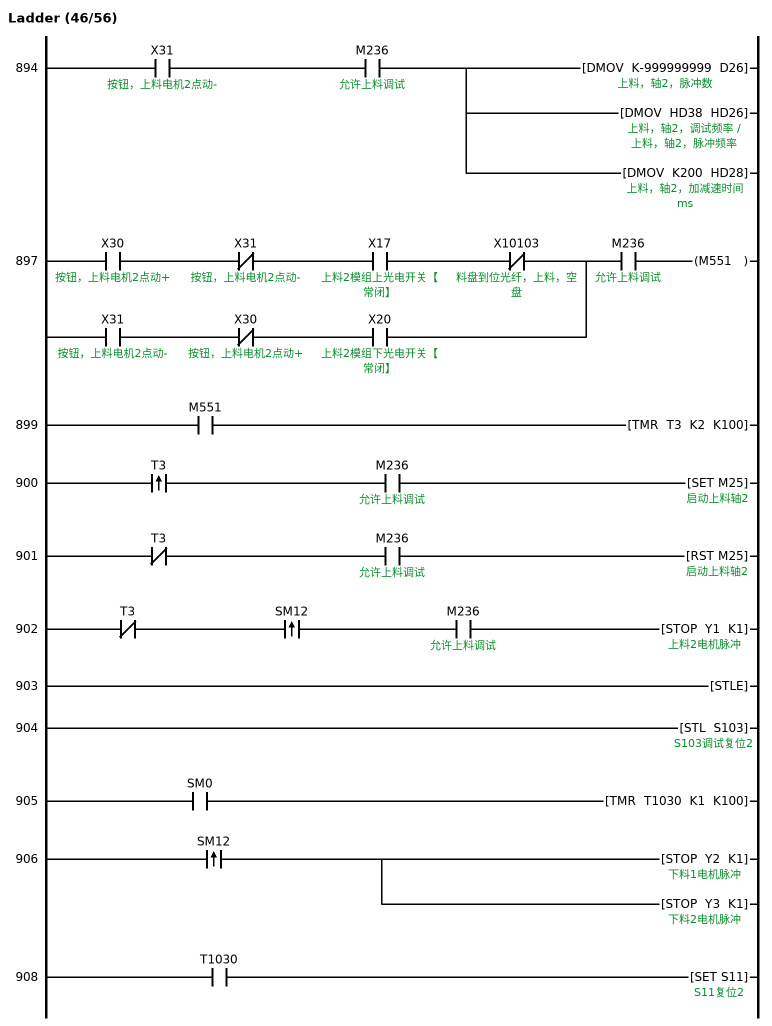
LD     X31	; 按钮，上料电机2点动-
AND    M236	; 允许上料调试
DMOV   K-999999999 D26	; 上料，轴2，脉冲数
DMOV   HD38 HD26	; 上料，轴2，调试频率 / 上料，轴2，脉冲频率
DMOV   K200 HD28	; 上料，轴2，加减速时间ms
LD     X30	; 按钮，上料电机2点动+
ANI    X31	; 按钮，上料电机2点动-
AND    X17	; 上料2模组上光电开关【常闭】
ANI    X10103	; 料盘到位光纤，上料，空盘
LD     X31	; 按钮，上料电机2点动-
ANI    X30	; 按钮，上料电机2点动+
AND    X20	; 上料2模组下光电开关【常闭】
ORB
AND    M236	; 允许上料调试
OUT    M551
LD     M551
TMR    T3 K2 K100
LDP    T3
AND    M236	; 允许上料调试
SET    M25	; 启动上料轴2
LDI    T3
AND    M236	; 允许上料调试
RST    M25	; 启动上料轴2
LDI    T3
ANDP   SM12
AND    M236	; 允许上料调试
STOP   Y1 K1	; 上料2电机脉冲
STLE
STL    S103	; S103调试复位2
LD     SM0
TMR    T1030 K1 K100
LDP    SM12
STOP   Y2 K1	; 下料1电机脉冲
STOP   Y3 K1	; 下料2电机脉冲
LD     T1030
SET    S11	; S11复位2

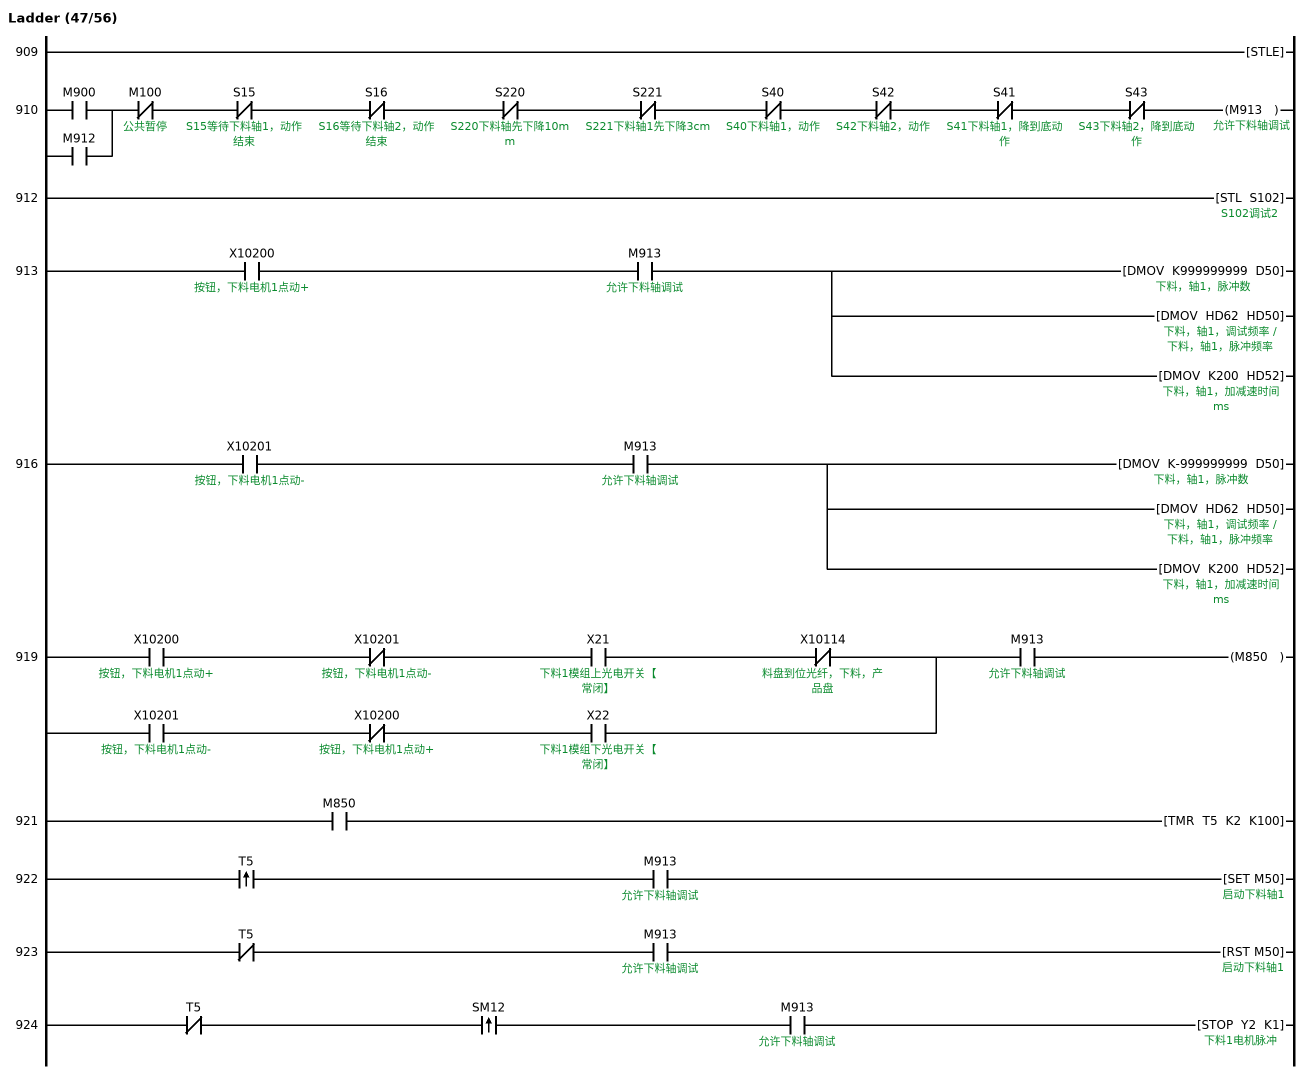
STLE
LD     M900
OR     M912
ANI    M100	; 公共暂停
ANI    S15	; S15等待下料轴1，动作结束
ANI    S16	; S16等待下料轴2，动作结束
ANI    S220	; S220下料轴先下降10mm
ANI    S221	; S221下料轴1先下降3cm
ANI    S40	; S40下料轴1，动作
ANI    S42	; S42下料轴2，动作
ANI    S41	; S41下料轴1，降到底动作
ANI    S43	; S43下料轴2，降到底动作
OUT    M913	; 允许下料轴调试
STL    S102	; S102调试2
LD     X10200	; 按钮，下料电机1点动+
AND    M913	; 允许下料轴调试
DMOV   K999999999 D50	; 下料，轴1，脉冲数
DMOV   HD62 HD50	; 下料，轴1，调试频率 / 下料，轴1，脉冲频率
DMOV   K200 HD52	; 下料，轴1，加减速时间ms
LD     X10201	; 按钮，下料电机1点动-
AND    M913	; 允许下料轴调试
DMOV   K-999999999 D50	; 下料，轴1，脉冲数
DMOV   HD62 HD50	; 下料，轴1，调试频率 / 下料，轴1，脉冲频率
DMOV   K200 HD52	; 下料，轴1，加减速时间ms
LD     X10200	; 按钮，下料电机1点动+
ANI    X10201	; 按钮，下料电机1点动-
AND    X21	; 下料1模组上光电开关【常闭】
ANI    X10114	; 料盘到位光纤，下料，产品盘
LD     X10201	; 按钮，下料电机1点动-
ANI    X10200	; 按钮，下料电机1点动+
AND    X22	; 下料1模组下光电开关【常闭】
ORB
AND    M913	; 允许下料轴调试
OUT    M850
LD     M850
TMR    T5 K2 K100
LDP    T5
AND    M913	; 允许下料轴调试
SET    M50	; 启动下料轴1
LDI    T5
AND    M913	; 允许下料轴调试
RST    M50	; 启动下料轴1
LDI    T5
ANDP   SM12
AND    M913	; 允许下料轴调试
STOP   Y2 K1	; 下料1电机脉冲

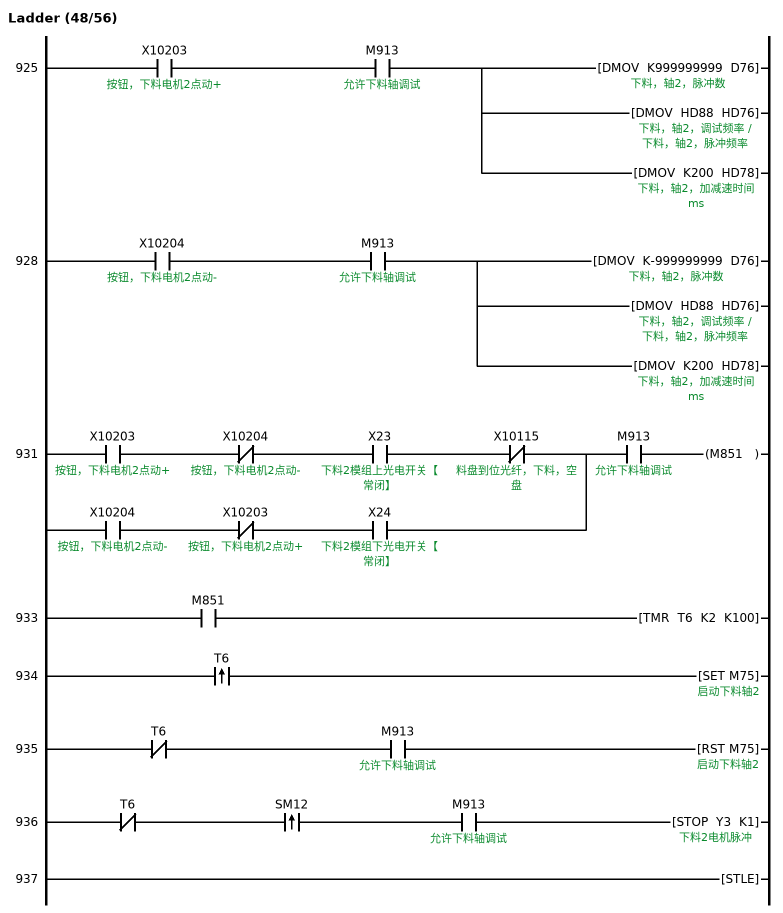
LD     X10203	; 按钮，下料电机2点动+
AND    M913	; 允许下料轴调试
DMOV   K999999999 D76	; 下料，轴2，脉冲数
DMOV   HD88 HD76	; 下料，轴2，调试频率 / 下料，轴2，脉冲频率
DMOV   K200 HD78	; 下料，轴2，加减速时间ms
LD     X10204	; 按钮，下料电机2点动-
AND    M913	; 允许下料轴调试
DMOV   K-999999999 D76	; 下料，轴2，脉冲数
DMOV   HD88 HD76	; 下料，轴2，调试频率 / 下料，轴2，脉冲频率
DMOV   K200 HD78	; 下料，轴2，加减速时间ms
LD     X10203	; 按钮，下料电机2点动+
ANI    X10204	; 按钮，下料电机2点动-
AND    X23	; 下料2模组上光电开关【常闭】
ANI    X10115	; 料盘到位光纤，下料，空盘
LD     X10204	; 按钮，下料电机2点动-
ANI    X10203	; 按钮，下料电机2点动+
AND    X24	; 下料2模组下光电开关【常闭】
ORB
AND    M913	; 允许下料轴调试
OUT    M851
LD     M851
TMR    T6 K2 K100
LDP    T6
SET    M75	; 启动下料轴2
LDI    T6
AND    M913	; 允许下料轴调试
RST    M75	; 启动下料轴2
LDI    T6
ANDP   SM12
AND    M913	; 允许下料轴调试
STOP   Y3 K1	; 下料2电机脉冲
STLE

